// TwinCAT 3 PLC project lcls_twincat_optics_plc
// Title: lcls-twincat-optics
// Company: SLAC
// ProjectVersion: 0.0.0
// ProgramVersion: 3.1.4022.3
// libraries:
//   LCLS General, * (SLAC)
//   Tc2_ControllerToolbox, * (Beckhoff Automation GmbH)
//   Tc2_MC2, * (Beckhoff Automation GmbH)
//   Tc2_SerialCom, * (Beckhoff Automation GmbH)
//   Tc2_Standard, * (Beckhoff Automation GmbH)
//   Tc2_System, * (Beckhoff Automation GmbH)
//   Tc2_Utilities, * (Beckhoff Automation GmbH)
//   Tc3_Module, * (Beckhoff Automation GmbH)
//   lcls-twincat-motion,1.1.0,SLAC
//   TcUnit,1.0.0.0,www.tcunit.org
// project tree:
//   DUTs/ DUT_HOMS.TcDUT (not stored), E_PiezoControl.TcDUT (not stored), E_PitchControl.TcDUT (not stored), HOMS_PitchMechanism.TcDUT (not stored), ST_PiezoAxis.TcDUT (not stored)
//   GVLs/ GVL_Constants.TcGVL (not stored), GVL_CoupledAfterStartup.TcGVL, GVL_DecoupledGantryDecrease.TcGVL, GVL_GantryInterlockStopsMotion.TcGVL
//   / PlcTask.TcTTO
//   POUs/ FB_Bender.TcPOU (not stored), FB_PiezoControl.TcPOU, FB_PitchControl.TcPOU (not stored), FB_RMSWatch.TcPOU, FB_RunHOMS.TcPOU, Main.TcPOU
//   POUs/Helpers/ FB_PI_E621_SerialDriver.TcPOU (not stored), FB_PI_E621_SerialTransaction.TcPOU (not stored), MC_SmoothMover.TcPOU (not stored), WithinRange.TcPOU (not stored)
//   POUs/Test/ FB_RunHOMS_Test.TcPOU, PRG_TEST.TcPOU, TEST_PitchControl.TcPOU (not stored)
//   Version/ Global_Version.TcGVL (not stored)
// real-time tasks:
//   TASK PlcTask: cycle T#10ms, priority 20, ADS port 350
// motion (NC):
//   TASK NC-Task 1 SAF: cycle T#2ms, priority 4, ADS port 501
//   TASK NC-Task 1 SVB: cycle T#10ms, priority 8, ADS port 511
//   AXIS TestAxisYup (id 2)
//     OtherSettings: AllowMotionCmdToSlave=true
//     encoder EncType=1
//     drive DrvType=5
//       Analog: ScaleFactorActTorque=0.1
//       TimeComp: TaskDelayCycles=1
//     controller CtrType=1
//       CtrPara: PriorControlFactor=1
//         Observer: BandWidth=20
//   AXIS TestAxisYdwn (id 8)
//     OtherSettings: AllowMotionCmdToSlave=true
//     encoder EncType=1
//     drive DrvType=5
//       Analog: ScaleFactorActTorque=0.1
//       TimeComp: TaskDelayCycles=1
//     controller CtrType=1
//       CtrPara: PriorControlFactor=1
//         Observer: BandWidth=20
//   AXIS TestAxisXup (id 9)
//     OtherSettings: AllowMotionCmdToSlave=true
//     encoder EncType=1
//     drive DrvType=5
//       Analog: ScaleFactorActTorque=0.1
//     controller CtrType=1
//       CtrPara: PriorControlFactor=1
//         Observer: BandWidth=20
//   AXIS TestAxisXdwn (id 10)
//     OtherSettings: AllowMotionCmdToSlave=true
//     encoder EncType=1
//     drive DrvType=5
//       Analog: ScaleFactorActTorque=0.1
//     controller CtrType=1
//       CtrPara: PriorControlFactor=1
//         Observer: BandWidth=20
//   AXIS TestAxisPitch (id 11)
//     OtherSettings: AllowMotionCmdToSlave=true
//     encoder EncType=1
//     drive DrvType=5
//       Analog: ScaleFactorActTorque=0.1
//     controller CtrType=1
//       CtrPara: PriorControlFactor=1
//         Observer: BandWidth=20
//   AXIS TestAxisMaster (id 12)
//     OtherSettings: AllowMotionCmdToSlave=true
//     encoder EncType=1
//     drive DrvType=5
//       Analog: ScaleFactorActTorque=0.1
//     controller CtrType=1
//       CtrPara: PriorControlFactor=1
//         Observer: BandWidth=20
//   AXIS TestAxisSlave (id 13)
//     OtherSettings: AllowMotionCmdToSlave=true
//     encoder EncType=1
//     drive DrvType=5
//       Analog: ScaleFactorActTorque=0.1
//     controller CtrType=1
//       CtrPara: PriorControlFactor=1
//         Observer: BandWidth=20
//   AXIS Axis 1 (id 1)
//     OtherSettings: AllowMotionCmdToSlave=true
//     encoder EncType=1
//     drive DrvType=5
//       Analog: ScaleFactorActTorque=0.1
//       TimeComp: TaskDelayCycles=1
//     controller CtrType=1
//       CtrPara: PriorControlFactor=1
//         Observer: BandWidth=20
//   AXIS Axis 2 (id 3)
//     OtherSettings: AllowMotionCmdToSlave=true
//     encoder EncType=1
//     drive DrvType=5
//       Analog: ScaleFactorActTorque=0.1
//       TimeComp: TaskDelayCycles=1
//     controller CtrType=1
//       CtrPara: PriorControlFactor=1
//         Observer: BandWidth=20
//   AXIS Axis 3 (id 4)
//     OtherSettings: AllowMotionCmdToSlave=true
//     encoder EncType=1
//     drive DrvType=5
//       Analog: ScaleFactorActTorque=0.1
//       TimeComp: TaskDelayCycles=1
//     controller CtrType=1
//       CtrPara: PriorControlFactor=1
//         Observer: BandWidth=20
//   AXIS Axis 4 (id 5)
//     OtherSettings: AllowMotionCmdToSlave=true
//     encoder EncType=1
//     drive DrvType=5
//       Analog: ScaleFactorActTorque=0.1
//       TimeComp: TaskDelayCycles=1
//     controller CtrType=1
//       CtrPara: PriorControlFactor=1
//         Observer: BandWidth=20
//   AXIS Axis 5 (id 6)
//     OtherSettings: AllowMotionCmdToSlave=true
//     encoder EncType=1
//     drive DrvType=5
//       Analog: ScaleFactorActTorque=0.1
//       TimeComp: TaskDelayCycles=1
//     controller CtrType=1
//       CtrPara: PriorControlFactor=1
//         Observer: BandWidth=20
//   AXIS Axis 6 (id 7)
//     OtherSettings: AllowMotionCmdToSlave=true
//     encoder EncType=1
//     drive DrvType=5
//       Analog: ScaleFactorActTorque=0.1
//       TimeComp: TaskDelayCycles=1
//     controller CtrType=1
//       CtrPara: PriorControlFactor=1
//         Observer: BandWidth=20
// variable links:
//   lcls_twincat_optics_plc Instance <-> NC-Task 1 SAF/Axes/TestAxisMaster
//     PlcTask Inputs/GVL_GantryInterlockStopsMotion.M1.Axis.NcToPlc <-> Outputs/ToPlc
//     PlcTask Outputs/GVL_GantryInterlockStopsMotion.M1.Axis.PlcToNc <-> Inputs/FromPlc
//   lcls_twincat_optics_plc Instance <-> NC-Task 1 SAF/Axes/TestAxisMasterDecoupled
//     PlcTask Inputs/GVL_DecoupledGantryDecrease.M1.Axis.NcToPlc <-> Outputs/ToPlc
//     PlcTask Outputs/GVL_DecoupledGantryDecrease.M1.Axis.PlcToNc <-> Inputs/FromPlc
//   lcls_twincat_optics_plc Instance <-> NC-Task 1 SAF/Axes/TestAxisPitch
//     PlcTask Inputs/GVL_CoupledAfterStartup.M5.Axis.NcToPlc <-> Outputs/ToPlc
//     PlcTask Outputs/GVL_CoupledAfterStartup.M5.Axis.PlcToNc <-> Inputs/FromPlc
//   lcls_twincat_optics_plc Instance <-> NC-Task 1 SAF/Axes/TestAxisSlave
//     PlcTask Inputs/GVL_GantryInterlockStopsMotion.M2.Axis.NcToPlc <-> Outputs/ToPlc
//     PlcTask Outputs/GVL_GantryInterlockStopsMotion.M2.Axis.PlcToNc <-> Inputs/FromPlc
//   lcls_twincat_optics_plc Instance <-> NC-Task 1 SAF/Axes/TestAxisSlaveDecoupled
//     PlcTask Inputs/GVL_DecoupledGantryDecrease.M2.Axis.NcToPlc <-> Outputs/ToPlc
//     PlcTask Outputs/GVL_DecoupledGantryDecrease.M2.Axis.PlcToNc <-> Inputs/FromPlc
//   lcls_twincat_optics_plc Instance <-> NC-Task 1 SAF/Axes/TestAxisXdwn
//     PlcTask Inputs/GVL_CoupledAfterStartup.M4.Axis.NcToPlc <-> Outputs/ToPlc
//     PlcTask Outputs/GVL_CoupledAfterStartup.M4.Axis.PlcToNc <-> Inputs/FromPlc
//   lcls_twincat_optics_plc Instance <-> NC-Task 1 SAF/Axes/TestAxisXup
//     PlcTask Inputs/GVL_CoupledAfterStartup.M3.Axis.NcToPlc <-> Outputs/ToPlc
//     PlcTask Outputs/GVL_CoupledAfterStartup.M3.Axis.PlcToNc <-> Inputs/FromPlc
//   lcls_twincat_optics_plc Instance <-> NC-Task 1 SAF/Axes/TestAxisYdwn
//     PlcTask Inputs/GVL_CoupledAfterStartup.M2.Axis.NcToPlc <-> Outputs/ToPlc
//     PlcTask Outputs/GVL_CoupledAfterStartup.M2.Axis.PlcToNc <-> Inputs/FromPlc
//   lcls_twincat_optics_plc Instance <-> NC-Task 1 SAF/Axes/TestAxisYup
//     PlcTask Inputs/GVL_CoupledAfterStartup.M1.Axis.NcToPlc <-> Outputs/ToPlc
//     PlcTask Outputs/GVL_CoupledAfterStartup.M1.Axis.PlcToNc <-> Inputs/FromPlc

CONFIGURATION lcls_twincat_optics_plc
    RESOURCE PLC ON TwinCAT3
        TASK PlcTask(INTERVAL := T#10ms, PRIORITY := 20);
        PROGRAM PRG_TEST WITH PlcTask : PRG_TEST;
    END_RESOURCE
END_CONFIGURATION

// ---- GVLs/GVL_CoupledAfterStartup.TcGVL
{attribute 'qualified_only'}
VAR_GLOBAL
	TestPitch_LimitSwitches : HOMS_PitchMechanism := (ReqPosLimHi:=2000,
		                                              ReqPosLimLo:=-2000,
		                                              diEncPosLimHi:=10768330,
		                                              diEncPosLimLo:=8141680);

	// Test Motors
	M1 : DUT_MotionStage;
	M2 : DUT_MotionStage;
	M3 : DUT_MotionStage;
	M4 : DUT_MotionStage;
	M5 : DUT_MotionStage;
	
	bFirstCycle : BOOL := TRUE;
END_VAR

// ---- GVLs/GVL_DecoupledGantryDecrease.TcGVL
{attribute 'qualified_only'}
VAR_GLOBAL
	// Test Motors
	M1 : DUT_MotionStage;
	M2 : DUT_MotionStage;
	
	// Test Encoders
	stMasterEnc : ST_RenishawAbsEnc;
	stSlaveEnc : ST_RenishawAbsEnc;

	bExecuteCoupleIn : BOOL;
	bExecuteDecoupleIn : BOOL;
	bGantryAlreadyCoupledOut : BOOL;
	nCycleCount : INT;
	fbAutoCouple : FB_GantryAutoCoupling;
END_VAR

// ---- GVLs/GVL_GantryInterlockStopsMotion.TcGVL
{attribute 'qualified_only'}
VAR_GLOBAL
	// Test Motors
	M1 : DUT_MotionStage;
	M2 : DUT_MotionStage;
	
	// Test Encoders
	stMasterEnc : ST_RenishawAbsEnc;
	stSlaveEnc : ST_RenishawAbsEnc;
END_VAR

// ---- POUs/Test/PRG_TEST.TcPOU
PROGRAM PRG_TEST
VAR
	fbRunHOMSTest : FB_RunHOMS_Test;
END_VAR

TcUnit.RUN();

END_PROGRAM

// ---- POUs/Test/FB_RunHOMS_Test.TcPOU
FUNCTION_BLOCK FB_RunHOMS_Test EXTENDS TcUnit.FB_TestSuite
VAR
END_VAR

CoupledAfterStartup();
//GantryInterlockStopsMotion();
DecoupledGantryDecrease();

METHOD CoupledAfterStartup
VAR
	// Test Struct
	TestHOMS : DUT_HOMS;

	bExpectedCoupleStatus : BOOL := TRUE;
	bActualCoupleStatus : BOOL;
END_VAR
// Testing automatic coupling of gantried Y and X axes
// Currently takes 1 additinal cycle for coupling to take effect after the command is sent
// Therefore need to wait one cycle before checking couple status
TEST('CoupledAfterStartup');

TestHOMS.fbRunHOMS(stYup:=GVL_CoupledAfterStartup.M1,
		  		   stYdwn:=GVL_CoupledAfterStartup.M2,
		           stXup:=GVL_CoupledAfterStartup.M3,
		           stXdwn:=GVL_CoupledAfterStartup.M4,
		           stPitch:=GVL_CoupledAfterStartup.M5,
		           nYupEncRef:=0,
		           nYdwnEncRef:=0,
		           nXupEncRef:=0,
		           nXdwnEncRef:=0,
		           bExecuteCoupleY:=TestHOMS.bExecuteCoupleY,
                   bExecuteCoupleX:=TestHOMS.bExecuteCoupleX,
		           bExecuteDecoupleY:=TestHOMS.bExecuteDecoupleY,
                   bExecuteDecoupleX:=TestHOMS.bExecuteDecoupleX,
                   bGantryAlreadyCoupledY=>TestHOMS.bGantryAlreadyCoupledY,
                   bGantryAlreadyCoupledX=>TestHOMS.bGantryAlreadyCoupledX,
                   nCurrGantryY=>TestHOMS.nCurrGantryY,
                   nCurrGantryX=>TestHOMS.nCurrGantryX);

bActualCoupleStatus := TestHOMS.bGantryAlreadyCoupledY AND TestHOMS.bGantryAlreadyCoupledX;
IF NOT GVL_CoupledAfterStartup.bFirstCycle THEN
	AssertEquals(Expected := bExpectedCoupleStatus,
	         	 Actual := bActualCoupleStatus,
			 	 Message := 'Either the Y or X gantry axes did not couple after startup');
	TEST_FINISHED();
END_IF;
GVL_CoupledAfterStartup.bFirstCycle := FALSE;
END_METHOD

METHOD DecoupledGantryDecrease
VAR
	nCurrGantry : LINT;
//	fbAutoCouple : FB_GantryAutoCoupling;

	fbMotionStage_master : FB_MotionStage;
	fbMotionStage_slave : FB_MotionStage;
	
	bExpectedResult : BOOL := TRUE;
	bActualResult : BOOL;
END_VAR
// Testing motion stop for decoupled gantried axes when gantry > gantry tol
// and that motion is allowed in directions that reduce the gantry
TEST('DecoupledGantryDecrease');

GVL_DecoupledGantryDecrease.nCycleCount := GVL_DecoupledGantryDecrease.nCycleCount + 1;

// EnableBits
GVL_DecoupledGantryDecrease.M1.bLimitForwardEnable := True; // Enable Limits
GVL_DecoupledGantryDecrease.M1.bLimitBackwardEnable := True;
GVL_DecoupledGantryDecrease.M1.bPowerSelf := True; // Enable Power
GVL_DecoupledGantryDecrease.M1.bHardwareEnable := True; // Enable STO
GVL_DecoupledGantryDecrease.M1.nCommand := 3; // Enable Motion Through PLC
GVL_DecoupledGantryDecrease.M1.nEnableMode := ENUM_StageEnableMode.ALWAYS;

GVL_DecoupledGantryDecrease.M2.bLimitForwardEnable := True; // Enable Limits
GVL_DecoupledGantryDecrease.M2.bLimitBackwardEnable := True;
GVL_DecoupledGantryDecrease.M2.bPowerSelf := True; // Enable Power
GVL_DecoupledGantryDecrease.M2.bHardwareEnable := True; // Enable STO
GVL_DecoupledGantryDecrease.M2.nCommand := 3; // Enable Motion Through PLC
GVL_DecoupledGantryDecrease.M2.nEnableMode := ENUM_StageEnableMode.ALWAYS;

// Enc Ref Vals
GVL_DecoupledGantryDecrease.stMasterEnc.Ref := 0;
GVL_DecoupledGantryDecrease.stSlaveEnc.Ref := 0;

// Fake Encoder Position Readback
GVL_DecoupledGantryDecrease.stMasterEnc.Count := 10000000 + LREAL_TO_ULINT(GVL_DecoupledGantryDecrease.M1.stAxisStatus.fActPosition * EXPT(10, 5)); // Position positive => counts up
GVL_DecoupledGantryDecrease.stSlaveEnc.Count := 10000000 + LREAL_TO_ULINT(GVL_DecoupledGantryDecrease.M2.stAxisStatus.fActPosition * EXPT(10, 5)); // Position negative => counts down

nCurrGantry := ((ULINT_TO_LINT(GVL_DecoupledGantryDecrease.stMasterEnc.Count) - ULINT_TO_LINT(GVL_DecoupledGantryDecrease.stMasterEnc.Ref)) - (ULINT_TO_LINT(GVL_DecoupledGantryDecrease.stSlaveEnc.Count) - ULINT_TO_LINT(GVL_DecoupledGantryDecrease.stSlaveEnc.Ref)));

IF GVL_DecoupledGantryDecrease.nCycleCount = 5 THEN
	GVL_DecoupledGantryDecrease.bExecuteDecoupleIn := TRUE;
	GVL_DecoupledGantryDecrease.M1.fPosition := 10.0;
	GVL_DecoupledGantryDecrease.M1.fVelocity := 0.2;

	GVL_DecoupledGantryDecrease.M2.fPosition := -10.0;
	GVL_DecoupledGantryDecrease.M2.fVelocity := 0.2;
END_IF;
	
IF GVL_DecoupledGantryDecrease.nCycleCount = 10 THEN
	GVL_DecoupledGantryDecrease.M1.bExecute := TRUE;
	GVL_DecoupledGantryDecrease.M2.bExecute := TRUE;
END_IF;

GVL_DecoupledGantryDecrease.fbAutoCouple(
	nGantryTol:=GVL_Constants.nGANTRY_TOLERANCE_NM_DEFAULT,
    Master:=GVL_DecoupledGantryDecrease.M1,
    MasterEnc:=GVL_DecoupledGantryDecrease.stMasterEnc,
    Slave:=GVL_DecoupledGantryDecrease.M2,
	SlaveEnc:=GVL_DecoupledGantryDecrease.stSlaveEnc,
    bExecuteCouple:=GVL_DecoupledGantryDecrease.bExecuteCoupleIn,
    bExecuteDecouple:=GVL_DecoupledGantryDecrease.bExecuteDecoupleIn,
	bGantryAlreadyCoupled=>GVL_DecoupledGantryDecrease.bGantryAlreadyCoupledOut);

fbMotionStage_master(stMotionStage:=GVL_DecoupledGantryDecrease.M1);
fbMotionStage_slave(stMotionStage:=GVL_DecoupledGantryDecrease.M2);

IF nCurrGantry > GVL_Constants.nGANTRY_TOLERANCE_NM_DEFAULT THEN
	bActualResult := (NOT GVL_DecoupledGantryDecrease.M1.bAllForwardEnable) AND (GVL_DecoupledGantryDecrease.M1.bAllBackwardEnable) AND (GVL_DecoupledGantryDecrease.M2.bAllForwardEnable) AND (NOT GVL_DecoupledGantryDecrease.M2.bAllBackwardEnable);
	AssertEquals(Expected := bExpectedResult,
		         Actual := bActualResult,
				 Message := 'Decoupled axes continued motion with gantry larger than the tolerance and/or motion not allowed in direction to reduce gantry');
	TEST_FINISHED();
END_IF;

IF GVL_DecoupledGantryDecrease.nCycleCount = 1000000000 THEN
	GVL_DecoupledGantryDecrease.nCycleCount := 0;
END_IF;
END_METHOD

METHOD GantryInterlockStopsMotion
VAR
	fEncSepFactor : REAL := 1.5;
	bExecuteCouple : BOOL;
	bExecuteDecouple : BOOL;
	bGantryAlreadyCoupled : BOOL;
	fbAutoCouple : FB_GantryAutoCoupling;
	fbMotionStage_master : FB_MotionStage;
	fbMotionStage_slave : FB_MotionStage;
	nCurrGantry : LINT;

	bExpectedEnableStatus : BOOL := FALSE;
	bActualEnableStatus : BOOL;
END_VAR
// Testing automatic motion stop when gantry difference of master and slave axes exceeds a tolerance
// Fake motor separation using fEncSepFactor which scales the readback of the master axis relative to the slave, causing the gantry to grow
// Ensuring Forward/Backward enables are FALSE for master and slave axes when gantry exceeds the tolerance
TEST('GantryInterlockStopsMotion');
// Cannot use FB_RunHOMS since enc counts are not inputs
// Need to test this behavior at next level down, i.e interfacing with fbAutoCouple

// Enable Bits
GVL_GantryInterlockStopsMotion.M1.bLimitForwardEnable := True; // Enable Limits
GVL_GantryInterlockStopsMotion.M1.bLimitBackwardEnable := True;
GVL_GantryInterlockStopsMotion.M1.bPowerSelf := True; // Enable Power
GVL_GantryInterlockStopsMotion.M1.bHardwareEnable := True; // Enable STO
GVL_GantryInterlockStopsMotion.M1.nCommand := 3; // Enable Motion Through PLC
GVL_GantryInterlockStopsMotion.M1.nEnableMode := ENUM_StageEnableMode.ALWAYS;

GVL_GantryInterlockStopsMotion.M2.bLimitForwardEnable := True; // Enable Limits
GVL_GantryInterlockStopsMotion.M2.bLimitBackwardEnable := True;
GVL_GantryInterlockStopsMotion.M2.bPowerSelf := True; // Enable Power
GVL_GantryInterlockStopsMotion.M2.bHardwareEnable := True; // Enable STO
GVL_GantryInterlockStopsMotion.M2.nCommand := 3; // Enable Motion Through PLC
GVL_GantryInterlockStopsMotion.M2.nEnableMode := ENUM_StageEnableMode.ALWAYS;

// Enc Ref Vals
GVL_GantryInterlockStopsMotion.stMasterEnc.Ref := 0;
GVL_GantryInterlockStopsMotion.stSlaveEnc.Ref := 0;

// Fake Encoder Position Readback
GVL_GantryInterlockStopsMotion.stMasterEnc.Count := LREAL_TO_ULINT(GVL_GantryInterlockStopsMotion.M1.stAxisStatus.fActPosition * fEncSepFactor * EXPT(10, 6));
GVL_GantryInterlockStopsMotion.stSlaveEnc.Count := LREAL_TO_ULINT(GVL_GantryInterlockStopsMotion.M2.stAxisStatus.fActPosition * EXPT(10, 6));

nCurrGantry := ((ULINT_TO_LINT(GVL_GantryInterlockStopsMotion.stMasterEnc.Count) - ULINT_TO_LINT(GVL_GantryInterlockStopsMotion.stMasterEnc.Ref)) - (ULINT_TO_LINT(GVL_GantryInterlockStopsMotion.stSlaveEnc.Count) - ULINT_TO_LINT(GVL_GantryInterlockStopsMotion.stSlaveEnc.Ref)));

fbAutoCouple(nGantryTol:=GVL_Constants.nGANTRY_TOLERANCE_NM_DEFAULT,
             Master:=GVL_GantryInterlockStopsMotion.M1,
             MasterEnc:=GVL_GantryInterlockStopsMotion.stMasterEnc,
             Slave:=GVL_GantryInterlockStopsMotion.M2,
	         SlaveEnc:=GVL_GantryInterlockStopsMotion.stSlaveEnc,
             bExecuteCouple:=bExecuteCouple,
             bExecuteDecouple:=bExecuteDecouple,
			 bGantryAlreadyCoupled=>bGantryAlreadyCoupled);

GVL_GantryInterlockStopsMotion.M1.fPosition := 5.0;
GVL_GantryInterlockStopsMotion.M1.fVelocity := 1.0;
GVL_GantryInterlockStopsMotion.M1.bExecute := TRUE;
	
fbMotionStage_master(stMotionStage:=GVL_GantryInterlockStopsMotion.M1);
fbMotionStage_slave(stMotionStage:=GVL_GantryInterlockStopsMotion.M2);

IF nCurrGantry > GVL_Constants.nGANTRY_TOLERANCE_NM_DEFAULT THEN
	bActualEnableStatus := (GVL_GantryInterlockStopsMotion.M1.bAllForwardEnable OR GVL_GantryInterlockStopsMotion.M1.bAllBackwardEnable OR GVL_GantryInterlockStopsMotion.M2.bAllForwardEnable OR GVL_GantryInterlockStopsMotion.M2.bAllBackwardEnable);
	AssertEquals(Expected := bExpectedEnableStatus,
		         Actual := bActualEnableStatus,
				 Message := 'Either master or slave continued motion after exceeding gantry tolerance');
	TEST_FINISHED();
END_IF;
END_METHOD

END_FUNCTION_BLOCK

// ---- POUs/FB_PiezoControl.TcPOU
FUNCTION_BLOCK FB_PiezoControl
VAR_IN_OUT
	iq_Piezo	:	ST_PiezoAxis;
END_VAR
VAR_INPUT
	xExecute	:	BOOL; //Rising edge being piezo motion
	xReset      :   BOOL;
	Enable_Positive : BOOL; //Reverse of Positive Limit Switch
	Enable_Negative : BOOL; //Reverse of Negative Limit Switch
END_VAR
VAR_OUTPUT
	xBusy	:	BOOL; //Busy remains true while piezo position is being adjusted
	xDone	:	BOOL; //Reached target position
	xError	:	BOOL; //General error
	xLimited:	BOOL; //Piezo move was limited
END_VAR
VAR
	E_State     : E_PiezoControl; //ENUM for Piezo Control State
	rtStartMove : R_TRIG; //Rising Trigger for Execution
	rtReset     : R_TRIG; //Rising Trigger for Error reset
	rSetpoint   : REAL;   //Internal Storage of Setpoint
	rReqVoltage	:	REAL; //requested voltage
	rLLSV: REAL := 0;
	rHLSV: REAL := 120;
	fbPI: FB_CTRL_PI;
	fbRamp: FB_CTRL_RAMP_GENERATOR_EXT;
	// FB initialized flag
	bInitialized: BOOL;
	//Get cycle time for control FBs
	fbGetCycleTime	:	FB_CTRL_GET_TASK_CYCLETIME;
	tTaskCycleTime: TIME;
	bCycleTimeValid: BOOL;
	rtVoltMode: R_TRIG;
	fOut: LREAL;
	fPiezoBias: LREAL := 60;
	fScale: REAL := -60;
	tonPiezoDone: TON := (PT:=T#2S);
	tonPiezoLimited: TON := (PT:=T#500MS);
	xVoltageLimited: BOOL;
	ftEnPos	:	F_TRIG;
	ftEnNeg	:	F_TRIG;
	rtEnPos	:	R_TRIG;
	rtEnNeg	:	R_TRIG;
	fOutLimitHolder	:	LREAL; //holds the limit value until restored
	fOutHiLimHolder	:	LREAL; //holds the limit value until restored
	fOutLoLimHolder	:	LREAL; //holds the limit value until restored
	xFirstPass 	: 	BOOL := TRUE;
END_VAR

// FB Piezo Control

//Triggers
///////////////////////////////
	rtStartMove(CLK:=xExecute);
	rtReset(CLK:=iq_Piezo.xEnable);
	rtVoltMode(CLK:=iq_Piezo.xVoltageMode);

//Status bits
///////////////////////////
xBusy S= rtStartMove.Q;
xDone R= rtStartMove.Q;
	
//Keep requested voltage to within limits
iq_Piezo.rReqVoltage := LIMIT(iq_Piezo.LowerVoltage, iq_Piezo.rReqVoltage, iq_Piezo.UpperVoltage);

//Limits
(* These appear flipped, but in-fact are not *)
ftEnPos(CLK:=Enable_Positive);
ftEnNeg(CLK:=Enable_Negative);
rtEnPos(CLK:=Enable_Positive);
rtEnNeg(CLK:=Enable_Negative);
IF xFirstPass THEN
	//Want to hold the limits on first pass if a switch is hit.
	(* When we move off the limit, we'll restore the init value (usually 1). This will be reset
	to something less than 1 when the limit gets tripped again, because presumably the actual limit
	would have been set at a value < 1 if the system had been runing.
	We just need to hold the init value to make it past this edge case that is present at startup. *)
	IF NOT Enable_Positive THEN fOutHiLimHolder := iq_Piezo.stPIParams.fOutMaxLimit; END_IF
	IF NOT Enable_Negative THEN fOutLoLimHolder := iq_Piezo.stPIParams.fOutMinLimit; END_IF
ELSE
	IF ftEnPos.Q THEN
		rLLSV := iq_Piezo.rSetVoltage;
		fOutHiLimHolder := iq_Piezo.stPIParams.fOutMaxLimit;
		iq_Piezo.stPIParams.fOutMaxLimit := fbPI.fOut;
	ELSIF rtEnPos.Q THEN
		rLLSV := iq_Piezo.LowerVoltage;
		iq_Piezo.stPIParams.fOutMaxLimit := fOutHiLimHolder;
	END_IF

	IF ftEnNeg.Q THEN
		rHLSV := iq_Piezo.rSetVoltage;
		
		fOutLoLimHolder := iq_Piezo.stPIParams.fOutMinLimit;
		iq_Piezo.stPIParams.fOutMinLimit := fbPI.fOut;
	ELSIF rtEnNeg.Q THEN
		rHLSV := iq_Piezo.UpperVoltage;
		iq_Piezo.stPIParams.fOutMinLimit := fOutLoLimHolder;
	END_IF
END_IF

// Don't do anything until we're ready
IF bInitialized THEN
	// While the block is working, a new position may be requested, this is OK
	IF xBusy THEN
		fbPI.fSetpointValue := iq_Piezo.rReqAbsPos;
	END_IF

	(* The next chunk of code prevents the PI block from winding up.
		First, when the PI block begins to request a voltage that is 
		beyond the permitted range (this range is affected by the state
		of limit switches/ or enable fwd/bwd), we latch the requested position.
		Presumeably this position request  *)

	//Select the PI block control mode
	////////////////////////////////////////
	IF iq_Piezo.xVoltageMode THEN
		//Set PI block to idle
		fbPI.eMode := eCTRL_MODE_PASSIVE;
		rReqVoltage := iq_Piezo.rReqVoltage; //TODO add a ramp
	ELSE
		IF iq_Piezo.xIdleMode THEN
			rReqVoltage := fScale * 0 + fPiezoBias;

			fbPI.eMode := eCTRL_MODE_MANUAL;
			ACT_Controller();
			fbPI.bHold := TRUE;
		ELSE
			//Fout is connected to the piezo voltage control
			rReqVoltage := fScale * fbPI.fOut + fPiezoBias;
			fbPI.bHold := FALSE;
			//Control mode is always active, so compensation takes over more smoothly
			fbPI.eMode := eCTRL_MODE_ACTIVE;
		END_IF		
	
	END_IF

	ACT_Controller();

	xVoltageLimited := rLLSV > rReqVoltage OR rHLSV < rReqVoltage;

	//This is where the voltage request gets sent to the piezo driver
	iq_Piezo.rSetVoltage := LIMIT(rLLSV, rReqVoltage, rHLSV);

//Initialization
ELSE
	fbGetCycleTime( eMode   := eCTRL_MODE_ACTIVE,
                tTaskCycleTime => tTaskCycleTime,
                bCycleTimeValid => bCycleTimeValid);
	IF bCycleTimeValid THEN
		iq_Piezo.stPIParams.tTaskCycleTime := tTaskCycleTime;
		iq_Piezo.stPIParams.tCtrlCycleTime := tTaskCycleTime;
		bInitialized	:= TRUE;
	END_IF

END_IF

tonPiezoDone.IN := WithinRange(ValA:=iq_Piezo.rActPos, Center:=iq_Piezo.rReqAbsPos, Range:=iq_Piezo.rPiezoDmovRange, Offset:=0) 
					AND NOT rtStartMove.Q; //rtStartMove interrupts the timer, resetting it
tonPiezoDone();

tonPiezoLimited.IN := (fbPI.bARWactive OR xVoltageLimited) AND NOT rtStartMove.Q;
tonPiezoLimited();

xDone S= xBusy AND (tonPiezoDone.Q OR tonPiezoLimited.Q);
xLimited := tonPiezoLimited.Q;

xBusy R= xDone;

xFirstPass := FALSE;

ACTION ACT_CheckLimits:

END_ACTION

ACTION ACT_Controller:
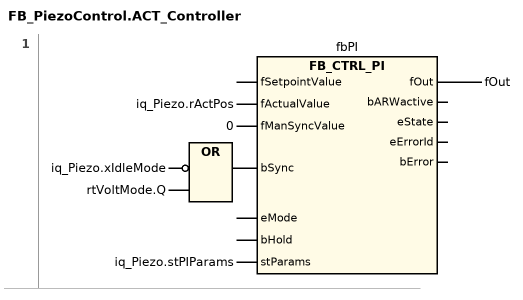
// NETWORK 1
fbPI(
    fActualValue := iq_Piezo.rActPos,
    fManSyncValue := 0,
    bSync := NOT iq_Piezo.xIdleMode OR rtVoltMode.Q,
    stParams := iq_Piezo.stPIParams); // FB_CTRL_PI
fOut := fbPI.fOut;
END_ACTION

END_FUNCTION_BLOCK

// ---- POUs/FB_RMSWatch.TcPOU
FUNCTION_BLOCK FB_RMSWatch
VAR_INPUT
END_VAR
VAR_OUTPUT
	// RMS Error
	fMaxRMSError : LREAL := 0;
	fMinRMSError : LREAL := 1000; // start at something huge, FB will update with any smaller measured value
END_VAR
VAR_IN_OUT
	stMotionStage : DUT_MotionStage;
END_VAR
VAR
	fbDataActPos : FB_LREALBuffer; // ActPos Data Acquisition FB
	fbDataSetPos : FB_LREALBuffer; // SetPos Data Acquisition FB
	bExecuteDataStorage : BOOL := TRUE; // Take data of both ActPos and SetPos
	bNewEncArray : BOOL;

	fbStats : FB_BasicStats; // Calculate mean/standard deviation of ActPos
	{attribute 'pytmc' := '
		pv: MEAN
		io: i
    '}
	fEncMean : LREAL;
	{attribute 'pytmc' := '
		pv: STDEV
		io: i
    '}
	fEncStDev : LREAL;
	{attribute 'pytmc' := '
		pv: RMS
		io: i
    '}
	fCurrRMSError : LREAL := 0;

	nIndex : DINT;
	fSum : LREAL := 0; // Just for calculating rms
	fDiff : LREAL := 0;

	{attribute 'pytmc' := '
		pv: ACTPOSARRAY
		io: i
    '}
	aEncActPos : ARRAY [1..1000] OF LREAL;
	{attribute 'pytmc' := '
		pv: SETPOSARRAY
		io: i
	'}
	aEncSetPos : ARRAY [1..1000] OF LREAL;
END_VAR

// FB to store encoder positions in 1000 element arrays, compute RMS errors, and watch for min/max

// Encoder Readback/Storage
fbDataActPos(bExecute:=bExecuteDataStorage,
           	 fInput:=stMotionStage.stAxisStatus.fActPosition,
           	 arrOutput=>aEncActPos,
             bNewArray=>bNewEncArray);

fbDataSetPos(bExecute:=bExecuteDataStorage,
           	 fInput:=stMotionStage.Axis.NcToPlc.SetPos,
           	 arrOutput=>aEncSetPos);

fbStats(aSignal:=aEncActPos,
	    bAlwaysCalc:=TRUE,
		fMean=>fEncMean,
		fStDev=>fEncStDev);

// Calculate RMS Error:
If bNewEncArray THEN
	fCurrRMSError := 0;
	FOR nIndex := 2 TO 1000 DO
		// First point in array stuck as 0 for some reason...
		fDiff := aEncActPos[nIndex] - aEncSetPos[nIndex];
		fSum := EXPT(fDiff, 2);
		fCurrRMSError := fCurrRMSError + fSum;
	END_FOR;
	fCurrRMSError := fCurrRMSError / 999.0; // 1000 element array but ditched the first point
	fCurrRMSError := SQRT(fCurrRMSError);
	// Watch for max:
	IF fCurrRMSError > fMaxRMSError THEN
		fMaxRMSError := fCurrRMSError;
	END_IF
	// Watch for min:
	IF fCurrRMSError < fMinRMSError THEN
		fMinRMSError := fCurrRMSError;
	END_IF
END_IF

END_FUNCTION_BLOCK

// ---- POUs/FB_RunHOMS.TcPOU
FUNCTION_BLOCK FB_RunHOMS
VAR_INPUT
	// Encoder Reference Values
	nYupEncRef : ULINT;
	nYdwnEncRef : ULINT;
	nXupEncRef : ULINT;
	nXdwnEncRef : ULINT;

	// Gantry Tolerances
	nGantryTolY : LINT := GVL_Constants.nGANTRY_TOLERANCE_NM_DEFAULT; // Encoder counts = nm
	nGantryTolX : LINT := GVL_Constants.nGANTRY_TOLERANCE_NM_DEFAULT; // Encoder counts = nm
END_VAR
VAR_OUTPUT
	// Gantry coupling status
	bGantryAlreadyCoupledY : BOOL;
	bGantryAlreadyCoupledX : BOOL;
	
	// Current gantry difference
	nCurrGantryY : LINT;
	nCurrGantryX : LINT;
END_VAR
VAR_IN_OUT
	// Motor Structs
	stYup : DUT_MotionStage;
	stYdwn : DUT_MotionStage;
	stXup : DUT_MotionStage;
	stXdwn : DUT_MotionStage;
	stPitch : DUT_MotionStage;

	// Manual coupling Gantried Axes
	bExecuteCoupleY : BOOL;
	bExecuteCoupleX : BOOL;
	bExecuteDecoupleY : BOOL;
	bExecuteDecoupleX : BOOL;
END_VAR
VAR
	// STO Button
	bSTOEnable1 AT %I* : BOOL;
	bSTOEnable2 AT %I* : BOOL;

	// Encoders
	stYupEnc AT %I* : ST_RenishawAbsEnc;
	stYdwnEnc AT %I* : ST_RenishawAbsEnc;
	
	stXupEnc AT %I* : ST_RenishawAbsEnc;
	stXdwnEnc AT %I* : ST_RenishawAbsEnc;

	// Autocoupling Gantried Axes
	fbAutoCoupleY : FB_GantryAutoCoupling;
	fbAutoCoupleX : FB_GantryAutoCoupling;
END_VAR

// Encoder Reference Values
stYupEnc.Ref := nYupEncRef;
stYdwnEnc.Ref := nYdwnEncRef;
stXupEnc.Ref := nXupEncRef;
stXdwnEnc.Ref := nXdwnEncRef;

// Gantry Differences to monitor
nCurrGantryY := ((ULINT_TO_LINT(stYupEnc.Count) - ULINT_TO_LINT(stYupEnc.Ref)) - (ULINT_TO_LINT(stYdwnEnc.Count) - ULINT_TO_LINT(stYdwnEnc.Ref)));
nCurrGantryX := ((ULINT_TO_LINT(stXupEnc.Count) - ULINT_TO_LINT(stXupEnc.Ref)) - (ULINT_TO_LINT(stXdwnEnc.Count) - ULINT_TO_LINT(stXdwnEnc.Ref)));

// Release the hounds!
stYup.bHardwareEnable := bSTOEnable1 AND bSTOEnable2;
stYdwn.bHardwareEnable := bSTOEnable1 AND bSTOEnable2;
stXup.bHardwareEnable := bSTOEnable1 AND bSTOEnable2;
stXdwn.bHardwareEnable := bSTOEnable1 AND bSTOEnable2;
stPitch.bHardwareEnable := bSTOEnable1 AND bSTOEnable2;

// Start Autocoupling
fbAutoCoupleY(nGantryTol:=nGantryTolY,
	          Master:=stYup,
			  MasterEnc:= stYupEnc,
			  Slave:=stYdwn,
			  SlaveEnc:=stYdwnEnc,
			  bExecuteCouple:=bExecuteCoupleY,
			  bExecuteDecouple:=bExecuteDecoupleY,
			  bGantryAlreadyCoupled=>bGantryAlreadyCoupledY);

fbAutoCoupleX(nGantryTol:=nGantryTolX,
	          Master:=stXup,
			  MasterEnc:= stXupEnc,
			  Slave:=stXdwn,
			  SlaveEnc:=stXdwnEnc,
			  bExecuteCouple:=bExecuteCoupleX,
			  bExecuteDecouple:=bExecuteDecoupleX,
			  bGantryAlreadyCoupled=>bGantryAlreadyCoupledX);

END_FUNCTION_BLOCK

// ---- POUs/Main.TcPOU
PROGRAM Main
VAR
	(*
	// Test Pitch Control
	fbPitchControl : FB_PitchControl;
	TestPitch : HOMS_PitchMechanism := (ReqPosLimHi:=2000,
		                                ReqPosLimLo:=-2000,
		                                diEncPosLimHi:=10768330,
		                                diEncPosLimLo:=8141680);
	M1 : DUT_MotionStage;
	bPitchDone : BOOL;
	*)

	// Test Bender vs No Bender
	TESTWithBender : DUT_HOMS;
	M1 : DUT_MotionStage := (nEnableMode:=ENUM_StageEnableMode.ALWAYS);
	M2 : DUT_MotionStage := (nEnableMode:=ENUM_StageEnableMode.ALWAYS);
	M3 : DUT_MotionStage := (nEnableMode:=ENUM_StageEnableMode.ALWAYS);
	M4 : DUT_MotionStage := (nEnableMode:=ENUM_StageEnableMode.ALWAYS);
	M5 : DUT_MotionStage := (nEnableMode:=ENUM_StageEnableMode.ALWAYS);
	M6 : DUT_MotionStage := (nEnableMode:=ENUM_StageEnableMode.ALWAYS);
	fbBender : FB_Bender;

	fbMotionStage_m1 : FB_MotionStage;
	fbMotionStage_m2 : FB_MotionStage;
	fbMotionStage_m3 : FB_MotionStage;
	fbMotionStage_m4 : FB_MotionStage;
	fbMotionStage_m6 : FB_MotionStage;
END_VAR

(*
// Test Pitch Control
M1.bLimitBackwardEnable;
M1.bLimitForwardEnable;
M1.bHardwareEnable;
M1.fVelocity := 150.0;
fbPitchControl(Pitch:=TestPitch,
			   Stepper:=M1,
			   lrCurrentSetpoint:=M1.fPosition,
			   q_bDone=>bPitchDone,
			   q_bBusy=>);
IF NOT M1.bHardwareEnable THEN
	M1.fPosition := M1.stAxisStatus.fActPosition;
END_IF
*)

// Test Bender vs. No Bender:
// M1L0
M1.bLimitForwardEnable := TRUE;
M1.bLimitBackwardEnable := TRUE;
M1.bPowerSelf := TRUE;

M2.bLimitForwardEnable := TRUE;
M2.bLimitBackwardEnable := TRUE;
M2.bPowerSelf := TRUE;

M3.bLimitForwardEnable := TRUE;
M3.bLimitBackwardEnable := TRUE;
M3.bPowerSelf := TRUE;

M4.bLimitForwardEnable := TRUE;
M4.bLimitBackwardEnable := TRUE;
M4.bPowerSelf := TRUE;

M5.bLimitForwardEnable := TRUE;
M5.bLimitBackwardEnable := TRUE;
M5.bPowerSelf := TRUE;

M6.bLimitForwardEnable := TRUE;
M6.bLimitBackwardEnable := TRUE;
M6.bPowerSelf := TRUE;
TESTWithBender.fbRunHOMS(stYup:=M1,
                         stYdwn:=M2,
                         stXup:=M3,
                         stXdwn:=M4,
                         stPitch:=M5,
	                     nYupEncRef:=0,
                         nYdwnEncRef:=0,
                         nXupEncRef:=0,
                         nXdwnEncRef:=0,
			             bExecuteCoupleY:=TESTWithBender.bExecuteCoupleY,
                         bExecuteCoupleX:=TESTWithBender.bExecuteCoupleX,
			             bExecuteDecoupleY:=TESTWithBender.bExecuteDecoupleY,
                         bExecuteDecoupleX:=TESTWithBender.bExecuteDecoupleX,
                         bGantryAlreadyCoupledY=>TESTWithBender.bGantryAlreadyCoupledY,
                         bGantryAlreadyCoupledX=>TESTWithBender.bGantryAlreadyCoupledX,
                         nCurrGantryY=>TESTWithBender.nCurrGantryY,
                         nCurrGantryX=>TESTWithBender.nCurrGantryX);
fbBender(stBender:=M6,
	     bSTOEnable1:=TESTWithBender.fbRunHOMS.bSTOEnable1,
		 bSTOEnable2:=TESTWithBender.fbRunHOMS.bSTOEnable2);

fbMotionStage_m1(stMotionStage:=M1);
fbMotionStage_m2(stMotionStage:=M2);
fbMotionStage_m3(stMotionStage:=M3);
fbMotionStage_m4(stMotionStage:=M4);
fbMotionStage_m6(stMotionStage:=M6);

END_PROGRAM
